Fanuc KAREL source: kd00072.KL

-- PROVISIONAL review KL for V770-1; original PC SHA256 1f1806c363d8f4aadc5e2f6d9259f34d8a9be02f6fa55a6a0a8b0cb40fb3f46f
-- Incomplete behavior may be omitted. Consult companion uncertainty JSON. Do not deploy.
PROGRAM KD00072
%NOLOCKGROUP
VAR
  I : INTEGER
  J : INTEGER
  B : BOOLEAN
  R : REAL
  S : STRING[80]
BEGIN
  -- UNRESOLVED_PC offsets 5-13; opcodes 9D,2E,1F
  -- UNRESOLVED_PC offsets 18-22; opcodes 7F
END KD00072
